// TIA Portal V19 export
DATA_BLOCK "DI_FW_HUB_links"   // DB22
AUTHOR : MS
// stored: AutoNumber false, InstanceOfName FB_HUB_FW_li, InstanceOfType FB
"FB_HUB_FW_li"
   // VAR_INPUT
   //    FW_DBNr : Int := 11;
   //    SysTime : Time := T#22M_15S_56MS;
   // END_VAR
   // VAR RETAIN
   //    Config : Struct
   //       Speed : Struct
   //          Min : Int := 5;
   //          Tipp : Int := 25;
   //          Hand : Int := 50;
   //          Max : Int := 100;
   //          Norm : Real := 0.0;
   //          endMess : Real := 0.0;
   //       END_STRUCT;
   //       Rampe : Struct
   //          Auf_Heben : Real := 0.0;
   //          Ab_Heben : Real := 0.0;
   //          Auf_Senken : Real := 0.0;
   //          Ab_Senken : Real := 0.0;
   //          NotStop : Real := 0.0;
   //       END_STRUCT;
   //       Bereich : Struct
   //          Pos : DInt := 10;
   //          Stop : DInt := 3;
   //          Ziel : DInt := 5;
   //          Absetzen : DInt := 300;
   //          Langsam : DInt := 200;
   //       END_STRUCT;
   //       TV_Position : DInt := 100;
   //       Reaktionszeit : Int := 0;
   //       Startzeit : Int := 0;
   //       Variante : Byte := 16#00;
   //       SimIstSpeed : Byte := 16#01;
   //       SimSensors : DWord := 16#4081_0102;
   //       SimTakt : DInt := 100;
   //    END_STRUCT;
   //    IN : Struct
   //       BA_Tipp : Bool := FALSE;
   //       BA_Hand : Bool := TRUE;
   //       BA_Auto : Bool := FALSE;
   //       Heben_aktiv : Bool := FALSE;
   //       Frg_Hub : Bool := FALSE;
   //       Frg_Eil : Bool := FALSE;
   //       Break_on : Bool := TRUE;
   //       mittig : Bool := FALSE;
   //       resB : Byte := 16#00;
   //       HubInc : DInt := 403;
   //       ZielInc : DInt := 0;
   //       Absetz_Inc : DInt := 400;
   //       IstSpeed : Int := 0;
   //    END_STRUCT;
   //    OUT : Struct
   //       Hub_Ok : Bool := TRUE;
   //       Break_off : Bool := FALSE;
   //       res_1 : Bool := FALSE;
   //       res_2 : Bool := FALSE;
   //       res_3 : Bool := FALSE;
   //       res_4 : Bool := FALSE;
   //       res_5 : Bool := FALSE;
   //       res_6 : Bool := FALSE;
   //       resB : Byte := 16#00;
   //       Bereich_langsam : DInt := 0;
   //       SollSpeed : Int := 0;
   //    END_STRUCT;
   //    Tmp : Struct
   //       lastTime : DInt := 1335056;
   //       DiffTime : Real := 10.0;
   //       lastSpeed : Real := 0.0;
   //       Messung : Struct
   //          lastInc : Real := 403.0;
   //          addInc : Real := 0.0;
   //          addTime : Real := 0.0;
   //          lastIst : Int := 0;
   //          messAct : Bool := FALSE;
   //       END_STRUCT;
   //       StopCount : DInt := 0;
   //       subInc : Real := 0.0;
   //       lastOut : Real := 0.0;
   //       TaktCount : Real := 0.0;
   //       PtrSensors : DWord := 16#0000_0001;
   //       RunTime : DInt := 0;
   //    END_STRUCT;
   // END_VAR
BEGIN
END_DATA_BLOCK
